TYPE EL4004_PDOS :
	STRUCT
		
		HwToPLC : EL4004_HWTOPLC_PDOS;
		
	END_STRUCT
END_TYPE

(* stored: Version 1.1.0.1
   DUT EL4004_PDOS: Id {f9edbe8c-4f47-48fe-b36b-4cddeea811cd} *)
